GLOBALCONSTANTS AID_AUXI2 (* Auxiliary input type 2 object attribute ids *)
  (* Standard: 61499-1; Description: Copyright (c) 2023 HR Agrartechnik GmbH This program and the accompanying materials are made available under the terms of the Eclipse Public License 2.0 which is available at https://www.eclipse.org/legal/epl-2.0/ SPDX-License-Identifier: EPL-2.0 *)
  (* Version 1.0, 2026-06-20, Franz Höpfinger, HR Agrartechnik GmbH *)
  PACKAGE isobus::UT::Q::const::AID;
  VAR_GLOBAL CONSTANT
    BACKGROUND_COLOUR : USINT := USINT#1; (* 1: AID_AUXI2_BACKGROUND_COLOUR - Background colour index. *)
    FUNC : USINT := USINT#2; (* 2: AID_AUXI2_FUNC (read-only) - Bitmask: Bits 0-4=Auxiliary function type (0-14), Bit 5=Critical Control, Bit *)
  END_VAR
END_GLOBALCONSTANTS
